(* IEC 61131-3 sources: IRIS-Project/LASAL CONTROL SOFTWARE/LasalProject_2025_09_12/Class/Motore_M2, 1 file *)

(* ---- Motore_M2.st ---- *)
(*!
<Class
	Name               = "Motore_M2"
	Revision           = "0.0"
	RealtimeTask       = "false"
	CyclicTask         = "true"
	DefCyclictime      = "100 ms"
	BackgroundTask     = "false"
	Sigmatek           = "false"
	OSInterface        = "false"
	HighPriority       = "false"
	Automatic          = "false"
	UpdateMode         = "Prescan"
	SharedCommandTable = "true"
	Objectsize         = "(720,180)">
	<Channels>
		<Server Name="ClassSvr" Visualized="false" Initialize="false" WriteProtected="true" Retentive="false"/>
		<Server Name="ErrorState" Visualized="false" Initialize="false" WriteProtected="true" Retentive="false"/>
		<Server Name="MotoreM2Step" Visualized="false" Initialize="false" WriteProtected="true" Retentive="false"/>
		<Server Name="s_1_3_pelletMode" Visualized="false" Initialize="false" WriteProtected="false" Retentive="false"/>
		<Server Name="s_M2_Homed" Visualized="false" Initialize="false" WriteProtected="false" Retentive="false"/>
		<Server Name="s_pelletInIrisCharge" Visualized="false" Initialize="false" WriteProtected="false" Retentive="false"/>
		<Server Name="s_tablet_InCharging" Visualized="false" Initialize="false" WriteProtected="false" Retentive="false"/>
		<Client Name="Comando_M2" Required="true" Internal="false"/>
		<Client Name="M2_LS" Required="false" Internal="false"/>
		<Client Name="SetPosition_Controller" Required="true" Internal="false"/>
	</Channels>
	<Separators>
		<Clients>
			<SepChn Position="1"/>
		</Clients>
	</Separators>
</Class>
*)
Motore_M2 : CLASS
	TYPE
	  t_sequence_Cmd_motore_M2 :  //! <Type Public="true" Name="t_sequence_Cmd_motore_M2"/>
	  (
	    Cmd_motore_M2_idle,
	    Cmd_motore_M2_homing,
	    Cmd_motore_M2_phasing,
	    Cmd_motore_M2_movement,
	    Cmd_motore_M2_reset,
	    Cmd_motore_M2_stop,
	    Cmd_motore_M2_stopped,
	    Cmd_motore_M2_Error
	  )$UDINT;
	END_TYPE
  //Servers:
	ClassSvr 	: SvrChCmd_DINT;
	MotoreM2Step 	: SvrCh_t_sequence_Cmd_motore_M2_PTofCls_Motore_M2;
	ErrorState 	: SvrCh__LMCAXIS_ERROR;
	s_M2_Homed 	: SvrCh_DINT;
	s_tablet_InCharging 	: SvrCh_DINT;
	s_1_3_pelletMode 	: SvrCh_DINT;
	s_pelletInIrisCharge 	: SvrCh_DINT;
  //Clients:
	Comando_M2 	: CltChCmd__LMCAxis;
	M2_LS 	: CltCh_DINT;
	SetPosition_Controller 	: CltCh_DINT;
  //Variables:
		ActCommand 	: t_sequence_Cmd_motore_M2;
		M2_homed 	: BOOL;
		Movement_step 	: DINT;
		M5_InPos 	: DINT;
		V_CONTATORE_TARGET_CARICATI 	: DINT;
		v_target_in_charge_slider 	: DINT;
		v_ErrorState 	: DINT;
		v_StartHomingCase 	: DINT;
		v_StartMovementCase 	: DINT;
		HomingStep 	: DINT;
		v_M2_LS 	: DINT;
		v_ACK_M1_No_Stuck_Mov 	: DINT;
		v_Req_No_Stuck_Mov_M1 	: DINT;
		v_AlternatingHoming 	: DINT;
		v_InCharging 	: DINT;
		v_PelletAvailable 	: DINT;
  //Functions:

	FUNCTION VIRTUAL GLOBAL Init;

	FUNCTION VIRTUAL GLOBAL CyWork
		VAR_INPUT
			EAX 	: UDINT;
		END_VAR
		VAR_OUTPUT
			state (EAX) 	: UDINT;
		END_VAR;

	FUNCTION GLOBAL SetSequenceState
		VAR_INPUT
			Cmd_motore 	: t_sequence_Cmd_motore_M2;
			StartCase 	: DINT;
		END_VAR
		VAR_OUTPUT
			retcode 	: DINT;
		END_VAR;

	FUNCTION GLOBAL GetHomedState
		VAR_OUTPUT
			Homed 	: BOOL;
		END_VAR;

	FUNCTION GLOBAL ReadM5PositionState
		VAR_INPUT
			Param 	: DINT;
		END_VAR;

	FUNCTION GLOBAL GetTargetInSlider
		VAR_OUTPUT
			Status 	: DINT;
		END_VAR;

	FUNCTION GLOBAL GetErrorState
		VAR_OUTPUT
			ErrorState 	: DINT;
		END_VAR;

	FUNCTION GLOBAL Req_M1_Mov
		VAR_OUTPUT
			OutParam 	: DINT;
		END_VAR;

	FUNCTION GLOBAL ACK_M1_Mov
		VAR_INPUT
			Param 	: DINT;
		END_VAR;

	FUNCTION GLOBAL GetPelletAvailable
		VAR_INPUT
			Param 	: DINT;
		END_VAR;

	FUNCTION VIRTUAL GLOBAL s_M2_Homed::Read
		VAR_OUTPUT
			output (EAX) 	: DINT;
		END_VAR;
  //Tables:
	FUNCTION @STD
		VAR_OUTPUT
			ret_code	: CONFSTATES;
		END_VAR;
	FUNCTION GLOBAL TAB @CT_;
END_CLASS;

#pragma usingLtd _LMCAxis

FUNCTION VIRTUAL GLOBAL Motore_M2::CyWork
	VAR_INPUT
		EAX 	: UDINT;
	END_VAR
	VAR_OUTPUT
		state (EAX) 	: UDINT;
	END_VAR

//M2: CHARGE BUFFER

  v_M2_LS:=M2_LS.Read();

  s_M2_Homed.Write(input:=M2_homed);

  case MotoreM2Step of
//===========================================================================================

    Cmd_motore_M2_idle:

    if Comando_M2.AxisError.HwError then
      v_ErrorState:=1;
      MotoreM2Step:=Cmd_motore_M2_Error;
    end_if;
//===========================================================================================

    Cmd_motore_M2_homing:

    // Si può pensare che la posizione di homing sia proprio quella di carica target poichè coincide con il tocco del LS

    if Comando_M2.AxisError.HwError then
      v_ErrorState:=1;
      HomingStep:=0;
      MotoreM2Step:=Cmd_motore_M2_Error;
    end_if;

    case HomingStep of

    0://idle
      HomingStep:=v_StartHomingCase;

    5:
      if v_M2_LS then //Motore già in posizione.
        HomingStep:=50;
      else
        HomingStep:=10;
      end_if;

    10://POER ON

      if (Comando_M2.AxisStatus.PowerOn=0) & (Comando_M2.AxisStatus.ReadyToPowerOn) then
        Comando_M2.PowerOn(Mode:=_LMCAXIS_MOVEDIRECTION::LMCAXIS_MOVE_ANY_WAY);
      elsif Comando_M2.AxisStatus.PowerOn then
        HomingStep:=20;
      end_if;

    20:
      Comando_M2.MoveEndless(Speed:=V_M2, Accel:=A_M2, Jerk:=J_M2);
      HomingStep:=30;

    30:
    if v_M2_LS then //quando tocca LS
      Comando_M2.StopMove(Decel:=A_M2, Jerk:=J_M2);
      HomingStep:=40;
    end_if;

    40://Controllo che il motore si sia fermato

      if Comando_M2.AxisStatus.Standstill then
          Comando_M2.PowerOff(Mode:=LMCAXIS_IMMEDIATE_STOPP);
          HomingStep:=50;
      end_if;

    50:
       if Comando_M2.AxisStatus.PowerOn=0 then
          M2_homed:=TRUE;
          SetPosition_Controller.Write(input:=0);
          MotoreM2Step:=Cmd_motore_M2_idle;
          v_StartHomingCase:=0;
       end_if;

    end_case;

//===========================================================================================

Cmd_motore_M2_movement:

    if Comando_M2.AxisError.HwError then
      v_ErrorState:=1;
      Movement_step:=0;
      MotoreM2Step:=Cmd_motore_M2_Error;
    end_if;

    case Movement_step of

      0: //IDLE, ATTESA COMANDI| Il motore è già nella posizione di carica->tocca il LS
        Movement_step:=v_StartMovementCase;

      10://M2 si trova nella posizione corretta di caricamento DEVE RUOTARE NEL VERSO CORRETTO PER SCARICARE TARGET, compirà 1 giro completo (quasi)
       if (Comando_M2.AxisStatus.PowerOn=0) & (Comando_M2.AxisStatus.ReadyToPowerOn) then
          Comando_M2.PowerOn(Mode:=LMCAXIS_MOVE_ANY_WAY);
       elsif Comando_M2.AxisStatus.PowerOn then
          if v_AlternatingHoming=1 then
            Movement_step:=20;
          elsif v_AlternatingHoming=-1 then
            Movement_step:=200;
          end_if;
        end_if;

      20:
		Comando_M2.MoveRelative(Position:=300000, Mode:=LMCAXIS_MOVE_RELATIVE_TO_POSITION, Speed:=V_M2, Accel:=A_M2, Decel:=A_M2, Jerk:=J_M2);
		Movement_step:=30;

      30:
		if Comando_M2.AxisStatus.InPosition & Comando_M2.AxisStatus.Standstill then
			Comando_M2.MoveAbsolute(Position:= 2300000, Speed:=V_M2, Accel:=A_M2, Decel:=A_M2, Jerk:=J_M2);
      s_pelletInIrisCharge.Write(input:=1);
      v_InCharging+=1;
			s_tablet_InCharging.Write(input:=v_InCharging);
			Movement_step:=40;
        end_if;

      40:
        if M2_LS.Read() | Comando_M2.AxisStatus.InPosition then
			v_target_in_charge_slider:=1;
			Comando_M2.StopMove(Decel:= A_M2, Jerk:= J_M2);
			Movement_step:=50;
        end_if;

	  50:
		if M5_InPos then
		    V_CONTATORE_TARGET_CARICATI+=1;
		    v_Req_No_Stuck_Mov_M1:=1;
		    v_target_in_charge_slider:=0;
		    Movement_step:=60;
		end_if;

      60://implementazione del movimento sù e giù dello scivolo per evitare lo stuck di un pellet
		if v_ACK_M1_No_Stuck_Mov then
			v_Req_No_Stuck_Mov_M1:=0;
			v_ACK_M1_No_Stuck_Mov:=0;
      v_InCharging+=1;
      s_pelletInIrisCharge.Write(input:=2);
			s_tablet_InCharging.Write(input:=v_InCharging);
		    if s_1_3_pelletMode.Read()=1 then //1 pellet
				Movement_step:=180;
			elsif s_1_3_pelletMode.Read()=0 then
				Movement_step:=70;
			end_if;
		end_if;

     70:
       Comando_M2.MoveRelative(Position:=- 300000, Mode:=LMCAXIS_MOVE_RELATIVE_TO_POSITION, Speed:=- V_M2, Accel:=- A_M2, Decel:=- A_M2, Jerk:=- J_M2);
       Movement_step:=80;

	    80:
       if Comando_M2.AxisStatus.InPosition & Comando_M2.AxisStatus.Standstill then
			    Comando_M2.MoveEndless(Speed:=- V_M2, Accel:=- A_M2, Jerk:=- J_M2);
          s_pelletInIrisCharge.Write(input:=3);
          v_InCharging+=1;
			    s_tablet_InCharging.Write(input:=v_InCharging);
			    Movement_step:=85;
       end_if;

     85:
       if M2_LS.Read() then
			    Comando_M2.StopMove(Decel:=- A_M2, Jerk:=- J_M2);
			    Movement_step:=86;
       end_if;

      86:
        Comando_M2.MoveRelative(Position:=- 50000, Mode:=LMCAXIS_MOVE_RELATIVE_TO_POSITION, Speed:=- V_M2, Accel:=- A_M2, Decel:=- A_M2, Jerk:=- J_M2);
        Movement_step:=90;

      90:
		    if Comando_M2.AxisStatus.InPosition & Comando_M2.AxisStatus.Standstill then
			      v_target_in_charge_slider:=1;
			      Comando_M2.StopMove(Decel:=-A_M2, Jerk:=-J_M2);
			      Movement_step:=100;
        end_if;

      100:
         if M5_InPos then
            V_CONTATORE_TARGET_CARICATI+=1;
            v_Req_No_Stuck_Mov_M1:=1;
            v_target_in_charge_slider:=0;
            Movement_step:=110;
         end_if;

      110://implementazione del movimento sù e giù dello scivolo per evitare lo stuck di un pellet

        if v_ACK_M1_No_Stuck_Mov then
          v_Req_No_Stuck_Mov_M1:=0;
          v_ACK_M1_No_Stuck_Mov:=0;
          s_pelletInIrisCharge.Write(input:=4);
          v_InCharging+=1;
          s_tablet_InCharging.Write(input:=v_InCharging);
          Movement_step:=120;
        end_if;

     120:
        Comando_M2.MoveRelative(Position:= 500000, Mode:=LMCAXIS_MOVE_RELATIVE_TO_POSITION, Speed:= V_M2, Accel:= A_M2, Decel:= A_M2, Jerk:= J_M2);
        Movement_step:=130;

     130:
        if Comando_M2.AxisStatus.InPosition & Comando_M2.AxisStatus.Standstill then
			      Comando_M2.MoveEndless(Speed:= V_M2, Accel:= A_M2, Jerk:= J_M2);
            s_pelletInIrisCharge.Write(input:=5);
            v_InCharging+=1;
			      s_tablet_InCharging.Write(input:=v_InCharging);
			      Movement_step:=140;
        end_if;

      140:
		     if M2_LS.Read() then
			      v_target_in_charge_slider:=1;
			      Comando_M2.StopMove(Decel:= A_M2, Jerk:= J_M2);
			      Movement_step:=150;
        end_if;

      145:
        Comando_M2.MoveRelative(Position:= 500000, Mode:=LMCAXIS_MOVE_RELATIVE_TO_POSITION, Speed:= V_M2, Accel:= A_M2, Decel:= A_M2, Jerk:= J_M2);
        Movement_step:=150;

      150:
         if M5_InPos then
            V_CONTATORE_TARGET_CARICATI+=1;
            v_Req_No_Stuck_Mov_M1:=1;
            v_target_in_charge_slider:=0;
            Movement_step:=160;
         end_if;

      160://implementazione del movimento sù e giù dello scivolo per evitare lo stuck di un pellet
        if v_ACK_M1_No_Stuck_Mov then
          v_Req_No_Stuck_Mov_M1:=0;
          v_ACK_M1_No_Stuck_Mov:=0;
          s_pelletInIrisCharge.Write(input:=6);
          v_InCharging+=1;
          s_tablet_InCharging.Write(input:=v_InCharging);
          Movement_step:=180;
        end_if;

      180:
        Comando_M2.PowerOff(Mode:=LMCAXIS_IMMEDIATE_STOPP);
        Movement_step:=190;

      190:
        if Comando_M2.AxisStatus.PowerOn=0 then
          v_AlternatingHoming:=-1*v_AlternatingHoming;
          v_StartMovementCase:=0;
          Movement_step:=0;
          MotoreM2Step:=Cmd_motore_M2_idle;
        end_if;

      200:
        Comando_M2.MoveRelative(Position:=-300000, Mode:=LMCAXIS_MOVE_RELATIVE_TO_POSITION, Speed:=-V_M2, Accel:=-A_M2, Decel:=-A_M2, Jerk:=-J_M2);
        Movement_step:=210;

      210:
        if Comando_M2.AxisStatus.InPosition & Comando_M2.AxisStatus.Standstill then
        	Comando_M2.MoveEndless(Speed:=-V_M2, Accel:=-A_M2, Jerk:=-J_M2);
          s_pelletInIrisCharge.Write(input:=1);
          v_InCharging+=1;
          s_tablet_InCharging.Write(input:=v_InCharging);
			    Movement_step:=220;
        end_if;

      220:
        if M2_LS.Read() | Comando_M2.AxisStatus.InPosition then
			    v_target_in_charge_slider:=1;
			    Comando_M2.StopMove(Decel:= -A_M2, Jerk:=-J_M2);
			    Movement_step:=230;
        end_if;

	    230:
			  if M5_InPos then
				  V_CONTATORE_TARGET_CARICATI+=1;
				  v_Req_No_Stuck_Mov_M1:=1;
				  v_target_in_charge_slider:=0;
				  Movement_step:=235;
			  end_if;

      235://implementazione del movimento sù e giù dello scivolo per evitare lo stuck di un pellet

        if v_ACK_M1_No_Stuck_Mov then
           v_Req_No_Stuck_Mov_M1:=0;
           v_ACK_M1_No_Stuck_Mov:=0;
           s_pelletInIrisCharge.Write(input:=2);
           v_InCharging+=1;
           s_tablet_InCharging.Write(input:=v_InCharging);
           if s_1_3_pelletMode.Read()=1 then //1 pellet
				      Movement_step:=340;
			     elsif s_1_3_pelletMode.Read()=0 then
				      Movement_step:=240;
			     end_if;

        end_if;

      240:
        Comando_M2.MoveRelative(Position:=300000, Mode:=LMCAXIS_MOVE_RELATIVE_TO_POSITION, Speed:=V_M2, Accel:=A_M2, Decel:=A_M2, Jerk:=J_M2);
        Movement_step:=250;

      250:
        if Comando_M2.AxisStatus.InPosition & Comando_M2.AxisStatus.Standstill then
        	Comando_M2.MoveEndless(Speed:=V_M2, Accel:=A_M2, Jerk:=J_M2);
          s_pelletInIrisCharge.Write(input:=3);
          v_InCharging+=1;
          s_tablet_InCharging.Write(input:=v_InCharging);
			    Movement_step:=260;
        end_if;

      260:
         if M2_LS.Read() then
          v_target_in_charge_slider:=1;
          Comando_M2.StopMove(Decel:=A_M2, Jerk:=J_M2);
          Movement_step:=270;
         end_if;

      270:
         if M5_InPos then
           V_CONTATORE_TARGET_CARICATI+=1;
           v_Req_No_Stuck_Mov_M1:=1;
           v_target_in_charge_slider:=0;
           Movement_step:=280;
         end_if;

      280://implementazione del movimento sù e giù dello scivolo per evitare lo stuck di un pellet

        if v_ACK_M1_No_Stuck_Mov then
           v_Req_No_Stuck_Mov_M1:=0;
           v_ACK_M1_No_Stuck_Mov:=0;
           s_pelletInIrisCharge.Write(input:=4);
           v_InCharging+=1;
           s_tablet_InCharging.Write(input:=v_InCharging);
           Movement_step:=290;
        end_if;

      290:
        Comando_M2.MoveRelative(Position:=-300000, Mode:=LMCAXIS_MOVE_RELATIVE_TO_POSITION, Speed:=-V_M2, Accel:=-A_M2, Decel:=-A_M2, Jerk:=-J_M2);
        Movement_step:=300;

      300:
        if Comando_M2.AxisStatus.InPosition & Comando_M2.AxisStatus.Standstill then
          Comando_M2.MoveEndless(Speed:=-V_M2, Accel:=-A_M2, Jerk:=-J_M2);
          s_pelletInIrisCharge.Write(input:=5);
          v_InCharging+=1;
          s_tablet_InCharging.Write(input:=v_InCharging);
			    Movement_step:=310;
        end_if;

      310:
        if M2_LS.Read() then
			    v_target_in_charge_slider:=1;
			    Comando_M2.StopMove(Decel:=-A_M2, Jerk:=-J_M2);
			    Movement_step:=320;
        end_if;

      320:
        if M5_InPos then
          V_CONTATORE_TARGET_CARICATI+=1;
          v_Req_No_Stuck_Mov_M1:=1;
          v_target_in_charge_slider:=0;
          Movement_step:=330;
        end_if;

      330://implementazione del movimento sù e giù dello scivolo per evitare lo stuck di un pellet
        if v_ACK_M1_No_Stuck_Mov then
           v_Req_No_Stuck_Mov_M1:=0;
           v_ACK_M1_No_Stuck_Mov:=0;
           s_pelletInIrisCharge.Write(input:=6);
           v_InCharging+=1;
           s_tablet_InCharging.Write(input:=v_InCharging);
           Movement_step:=340;
        end_if;

      340:
        Comando_M2.PowerOff(Mode:=LMCAXIS_IMMEDIATE_STOPP);
        Movement_step:=190;

    end_case;

//===========================================================================================

    Cmd_motore_M2_Error:

      ErrorState:=Comando_M2.AxisError; //AGGIORNAMENTO SERVER
      MotoreM2Step:=Cmd_motore_M2_stop;
//===========================================================================================

    Cmd_motore_M2_stop:

      if Comando_M2.AxisStatus.Standstill & Comando_M2.AxisStatus.PowerOn=0 then
        MotoreM2Step:=Cmd_motore_M2_stopped;
      else
        Comando_M2.QuickStop(Decel:=1000000);//se asse in errore non esegue neppure l'operazione perchè spento (e in errore)
        Comando_M2.PowerOff(Mode:=LMCAXIS_IMMEDIATE_STOPP);
      end_if;
//===========================================================================================

    Cmd_motore_M2_stopped:
    //ATTESA RESET
//===========================================================================================

    Cmd_motore_M2_reset:

      Comando_M2.QuitError();
      M2_homed:=FALSE;
      v_ErrorState:=0;
      if Comando_M2.AxisStatus.FiltRdy then
        MotoreM2Step:=Cmd_motore_M2_idle;
      end_if;

      Movement_step:=0;
      M5_InPos:=0;
      v_M2_LS:=0;
      v_ACK_M1_No_Stuck_Mov:=0;
      v_target_in_charge_slider:=0;
      v_StartHomingCase:=0;
      v_StartMovementCase:=0;
      HomingStep:=0;
      v_ErrorState:=0;
      s_pelletInIrisCharge.Write(input:=0);
      //s_1_3_pelletMode.Write(input:=0);

      if v_PelletAvailable<=V_CONTATORE_TARGET_CARICATI then
        s_tablet_InCharging.Write(input:=0);
        v_InCharging:=0;
        V_CONTATORE_TARGET_CARICATI:=0;
      end_if;

//===========================================================================================
  end_case;

	state := READY;
END_FUNCTION

FUNCTION GLOBAL Motore_M2::SetSequenceState
	VAR_INPUT
		Cmd_motore 	: t_sequence_Cmd_motore_M2;
		StartCase 	: DINT;
	END_VAR
	VAR_OUTPUT
		retcode 	: DINT;
	END_VAR

  if Cmd_motore=Cmd_motore_M2_homing then
    v_StartHomingCase:=StartCase;
  elsif Cmd_motore=Cmd_motore_M2_movement then
    v_StartMovementCase:=StartCase;
  end_if;

  MotoreM2Step:=Cmd_motore;
  retcode:=true;
END_FUNCTION

FUNCTION VIRTUAL GLOBAL Motore_M2::Init
M2_homed:=FALSE;
Movement_step:=0;
M5_InPos:=0;
v_M2_LS:=0;

v_ACK_M1_No_Stuck_Mov:=0;

V_CONTATORE_TARGET_CARICATI:=0;
v_target_in_charge_slider:=0;

v_StartHomingCase:=0;
v_StartMovementCase:=0;

HomingStep:=0;

v_ErrorState:=0;

v_AlternatingHoming:=1;

v_InCharging:=0;

v_PelletAvailable:=0;

END_FUNCTION

FUNCTION GLOBAL Motore_M2::GetHomedState
	VAR_OUTPUT
		Homed 	: BOOL;
	END_VAR

  Homed:=M2_homed;
END_FUNCTION

FUNCTION GLOBAL Motore_M2::ReadM5PositionState
	VAR_INPUT
		Param 	: DINT;
	END_VAR

  M5_InPos:=Param;
END_FUNCTION

FUNCTION GLOBAL Motore_M2::GetTargetInSlider
	VAR_OUTPUT
		Status 	: DINT;
	END_VAR

//v_target_in_charge_slider:=Status;
Status:=v_target_in_charge_slider;

END_FUNCTION

FUNCTION GLOBAL Motore_M2::GetErrorState
	VAR_OUTPUT
		ErrorState 	: DINT;
	END_VAR

  ErrorState:=v_ErrorState;

END_FUNCTION

FUNCTION VIRTUAL GLOBAL Motore_M2::s_M2_Homed::Read
	VAR_OUTPUT
		output (EAX) 	: DINT;
	END_VAR

	output := s_M2_Homed;

END_FUNCTION

FUNCTION GLOBAL Motore_M2::Req_M1_Mov
	VAR_OUTPUT
		OutParam 	: DINT;
	END_VAR
  OutParam:=v_Req_No_Stuck_Mov_M1;
END_FUNCTION

FUNCTION GLOBAL Motore_M2::ACK_M1_Mov
	VAR_INPUT
		Param 	: DINT;
	END_VAR
  v_ACK_M1_No_Stuck_Mov:=Param;
END_FUNCTION

FUNCTION GLOBAL Motore_M2::GetPelletAvailable
	VAR_INPUT
		Param 	: DINT;
	END_VAR
v_PelletAvailable:=Param;
END_FUNCTION
